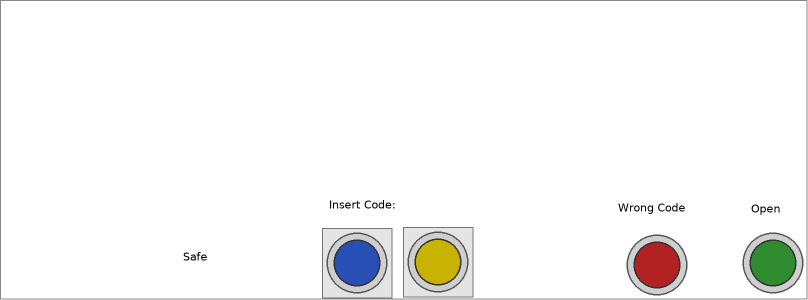
VISUALIZATION Visualization_Safe  // 808x300
    Label (326,190 147x30), "Insert Code:"
    Lamp1 (622,230 70x70), variable: GVL_IO.DO_LampRed, style: Lamp-Lamp1-Red
    PushSwitch (322,228 70x70), variable: GVL_IO.DI_BtnBlue, behaviour: TOGGLE, style: Switch-PushSwitch-Blue
    Lamp1 (738,228 70x70), variable: GVL_IO.DO_LampGreen, style: Lamp-Lamp1-Green
    PushSwitch (403,227 70x70), variable: GVL_IO.DI_BtnYellow, behaviour: TOGGLE, style: Switch-PushSwitch-Yellow
    Label (180,236 59x42), "Safe"
    Label (730,194 72x30), "Open"
    Label (616,193 72x30), "Wrong Code"
END_VISUALIZATION

(* stored: Version 1.1.0.1, ProductVersion 3.1.4024.9
   Visu Visualization_Safe: Id {56589513-9c75-4707-a394-0dfcb8a3f766} *)
